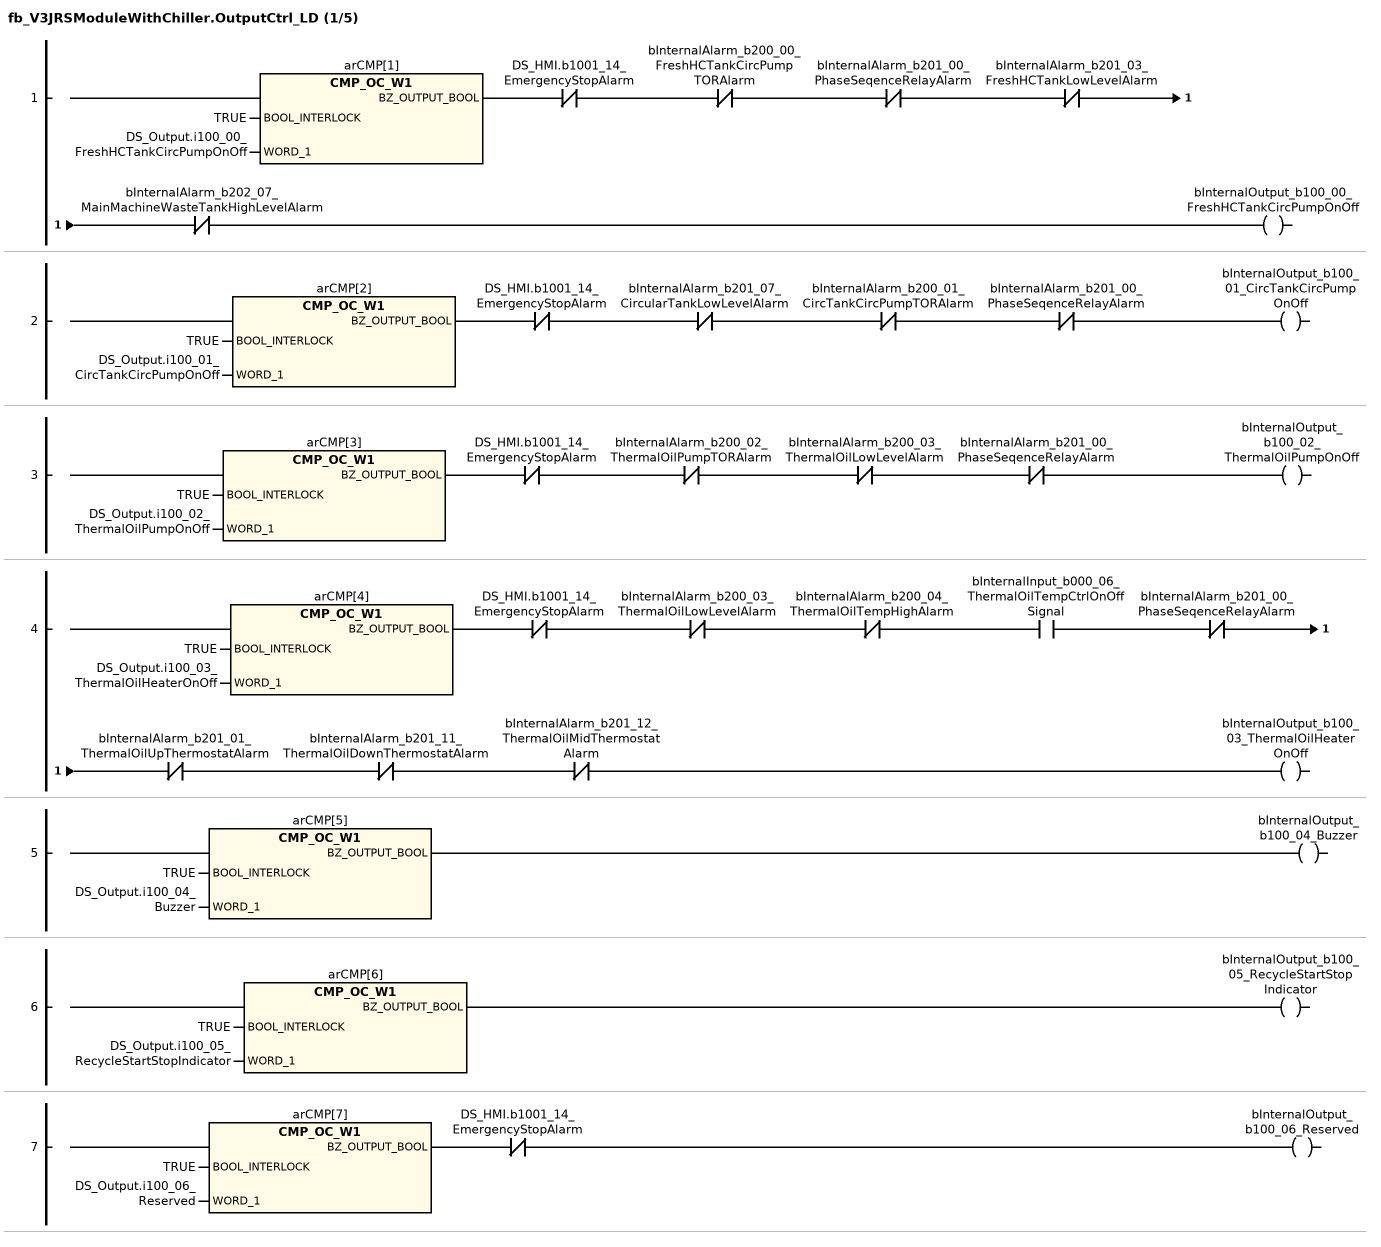
// NETWORK 1
arCMP[1](BOOL_INTERLOCK := TRUE, WORD_1 := DS_Output.i100_00_FreshHCTankCircPumpOnOff); // CMP_OC_W1
bInternalOutput_b100_00_FreshHCTankCircPumpOnOff := arCMP[1].BZ_OUTPUT_BOOL AND NOT DS_HMI.b1001_14_EmergencyStopAlarm AND NOT bInternalAlarm_b200_00_FreshHCTankCircPumpTORAlarm AND NOT bInternalAlarm_b201_00_PhaseSeqenceRelayAlarm AND NOT bInternalAlarm_b201_03_FreshHCTankLowLevelAlarm AND NOT bInternalAlarm_b202_07_MainMachineWasteTankHighLevelAlarm;

// NETWORK 2
arCMP[2](BOOL_INTERLOCK := TRUE, WORD_1 := DS_Output.i100_01_CircTankCircPumpOnOff); // CMP_OC_W1
bInternalOutput_b100_01_CircTankCircPumpOnOff := arCMP[2].BZ_OUTPUT_BOOL AND NOT DS_HMI.b1001_14_EmergencyStopAlarm AND NOT bInternalAlarm_b201_07_CircularTankLowLevelAlarm AND NOT bInternalAlarm_b200_01_CircTankCircPumpTORAlarm AND NOT bInternalAlarm_b201_00_PhaseSeqenceRelayAlarm;

// NETWORK 3
arCMP[3](BOOL_INTERLOCK := TRUE, WORD_1 := DS_Output.i100_02_ThermalOilPumpOnOff); // CMP_OC_W1
bInternalOutput_b100_02_ThermalOilPumpOnOff := arCMP[3].BZ_OUTPUT_BOOL AND NOT DS_HMI.b1001_14_EmergencyStopAlarm AND NOT bInternalAlarm_b200_02_ThermalOilPumpTORAlarm AND NOT bInternalAlarm_b200_03_ThermalOilLowLevelAlarm AND NOT bInternalAlarm_b201_00_PhaseSeqenceRelayAlarm;

// NETWORK 4
arCMP[4](BOOL_INTERLOCK := TRUE, WORD_1 := DS_Output.i100_03_ThermalOilHeaterOnOff); // CMP_OC_W1
bInternalOutput_b100_03_ThermalOilHeaterOnOff := arCMP[4].BZ_OUTPUT_BOOL AND NOT DS_HMI.b1001_14_EmergencyStopAlarm AND NOT bInternalAlarm_b200_03_ThermalOilLowLevelAlarm AND NOT bInternalAlarm_b200_04_ThermalOilTempHighAlarm AND bInternalInput_b000_06_ThermalOilTempCtrlOnOffSignal AND NOT bInternalAlarm_b201_00_PhaseSeqenceRelayAlarm AND NOT bInternalAlarm_b201_01_ThermalOilUpThermostatAlarm AND NOT bInternalAlarm_b201_11_ThermalOilDownThermostatAlarm AND NOT bInternalAlarm_b201_12_ThermalOilMidThermostatAlarm;

// NETWORK 5
arCMP[5](BOOL_INTERLOCK := TRUE, WORD_1 := DS_Output.i100_04_Buzzer); // CMP_OC_W1
bInternalOutput_b100_04_Buzzer := arCMP[5].BZ_OUTPUT_BOOL;

// NETWORK 6
arCMP[6](BOOL_INTERLOCK := TRUE, WORD_1 := DS_Output.i100_05_RecycleStartStopIndicator); // CMP_OC_W1
bInternalOutput_b100_05_RecycleStartStopIndicator := arCMP[6].BZ_OUTPUT_BOOL;

// NETWORK 7
arCMP[7](BOOL_INTERLOCK := TRUE, WORD_1 := DS_Output.i100_06_Reserved); // CMP_OC_W1
bInternalOutput_b100_06_Reserved := arCMP[7].BZ_OUTPUT_BOOL AND NOT DS_HMI.b1001_14_EmergencyStopAlarm;

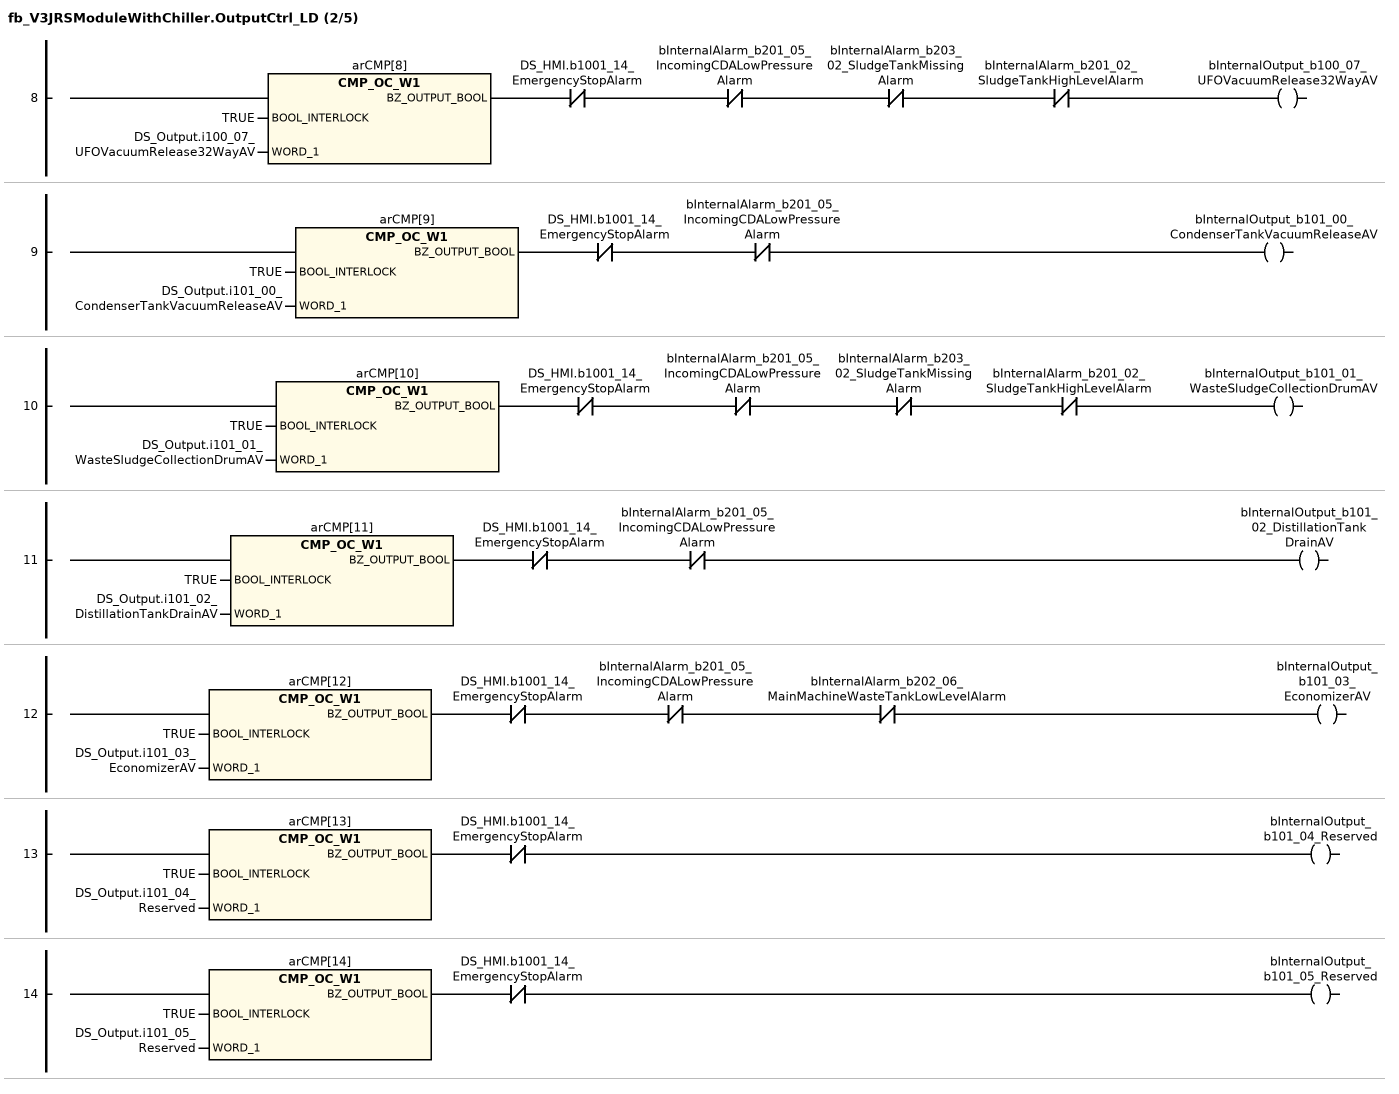
// NETWORK 8
arCMP[8](BOOL_INTERLOCK := TRUE, WORD_1 := DS_Output.i100_07_UFOVacuumRelease32WayAV); // CMP_OC_W1
bInternalOutput_b100_07_UFOVacuumRelease32WayAV := arCMP[8].BZ_OUTPUT_BOOL AND NOT DS_HMI.b1001_14_EmergencyStopAlarm AND NOT bInternalAlarm_b201_05_IncomingCDALowPressureAlarm AND NOT bInternalAlarm_b203_02_SludgeTankMissingAlarm AND NOT bInternalAlarm_b201_02_SludgeTankHighLevelAlarm;

// NETWORK 9
arCMP[9](BOOL_INTERLOCK := TRUE, WORD_1 := DS_Output.i101_00_CondenserTankVacuumReleaseAV); // CMP_OC_W1
bInternalOutput_b101_00_CondenserTankVacuumReleaseAV := arCMP[9].BZ_OUTPUT_BOOL AND NOT DS_HMI.b1001_14_EmergencyStopAlarm AND NOT bInternalAlarm_b201_05_IncomingCDALowPressureAlarm;

// NETWORK 10
arCMP[10](BOOL_INTERLOCK := TRUE, WORD_1 := DS_Output.i101_01_WasteSludgeCollectionDrumAV); // CMP_OC_W1
bInternalOutput_b101_01_WasteSludgeCollectionDrumAV := arCMP[10].BZ_OUTPUT_BOOL AND NOT DS_HMI.b1001_14_EmergencyStopAlarm AND NOT bInternalAlarm_b201_05_IncomingCDALowPressureAlarm AND NOT bInternalAlarm_b203_02_SludgeTankMissingAlarm AND NOT bInternalAlarm_b201_02_SludgeTankHighLevelAlarm;

// NETWORK 11
arCMP[11](BOOL_INTERLOCK := TRUE, WORD_1 := DS_Output.i101_02_DistillationTankDrainAV); // CMP_OC_W1
bInternalOutput_b101_02_DistillationTankDrainAV := arCMP[11].BZ_OUTPUT_BOOL AND NOT DS_HMI.b1001_14_EmergencyStopAlarm AND NOT bInternalAlarm_b201_05_IncomingCDALowPressureAlarm;

// NETWORK 12
arCMP[12](BOOL_INTERLOCK := TRUE, WORD_1 := DS_Output.i101_03_EconomizerAV); // CMP_OC_W1
bInternalOutput_b101_03_EconomizerAV := arCMP[12].BZ_OUTPUT_BOOL AND NOT DS_HMI.b1001_14_EmergencyStopAlarm AND NOT bInternalAlarm_b201_05_IncomingCDALowPressureAlarm AND NOT bInternalAlarm_b202_06_MainMachineWasteTankLowLevelAlarm;

// NETWORK 13
arCMP[13](BOOL_INTERLOCK := TRUE, WORD_1 := DS_Output.i101_04_Reserved); // CMP_OC_W1
bInternalOutput_b101_04_Reserved := arCMP[13].BZ_OUTPUT_BOOL AND NOT DS_HMI.b1001_14_EmergencyStopAlarm;

// NETWORK 14
arCMP[14](BOOL_INTERLOCK := TRUE, WORD_1 := DS_Output.i101_05_Reserved); // CMP_OC_W1
bInternalOutput_b101_05_Reserved := arCMP[14].BZ_OUTPUT_BOOL AND NOT DS_HMI.b1001_14_EmergencyStopAlarm;

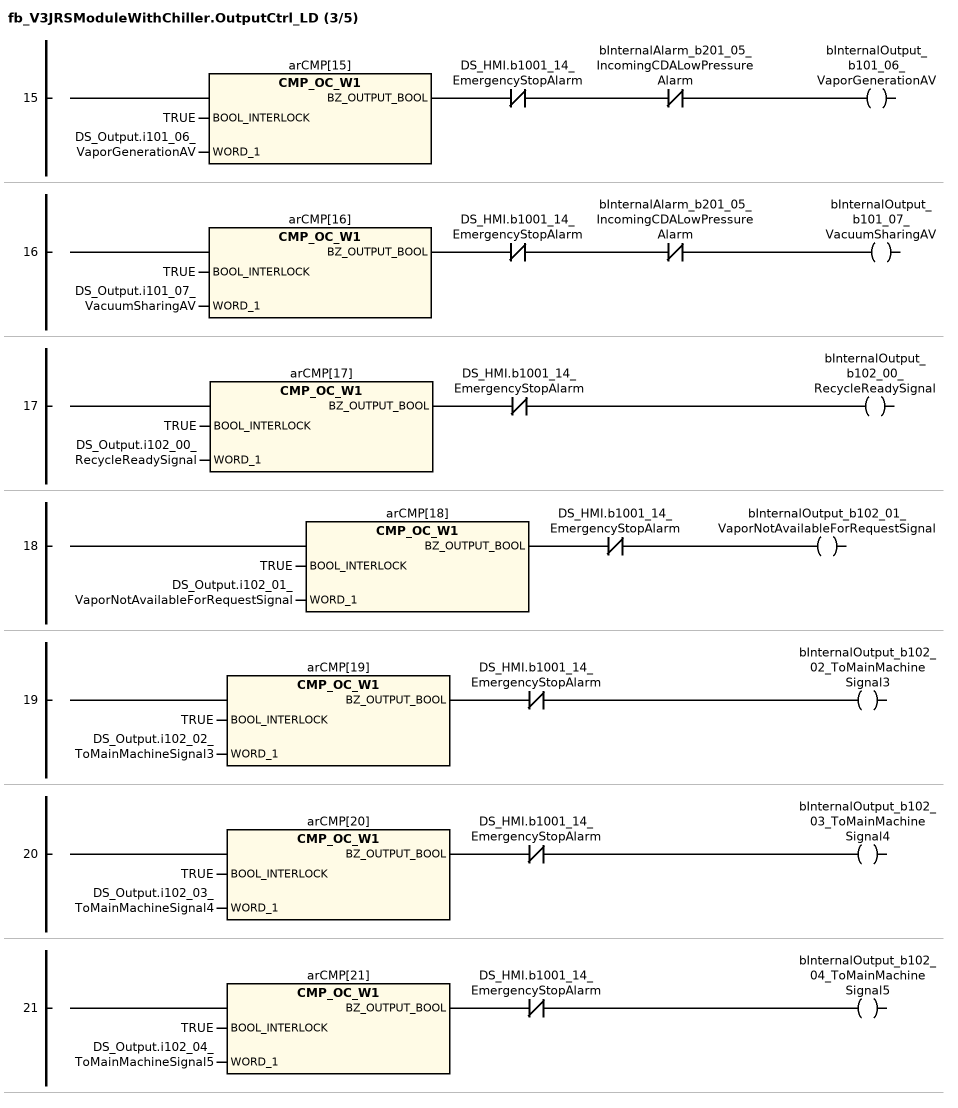
// NETWORK 15
arCMP[15](BOOL_INTERLOCK := TRUE, WORD_1 := DS_Output.i101_06_VaporGenerationAV); // CMP_OC_W1
bInternalOutput_b101_06_VaporGenerationAV := arCMP[15].BZ_OUTPUT_BOOL AND NOT DS_HMI.b1001_14_EmergencyStopAlarm AND NOT bInternalAlarm_b201_05_IncomingCDALowPressureAlarm;

// NETWORK 16
arCMP[16](BOOL_INTERLOCK := TRUE, WORD_1 := DS_Output.i101_07_VacuumSharingAV); // CMP_OC_W1
bInternalOutput_b101_07_VacuumSharingAV := arCMP[16].BZ_OUTPUT_BOOL AND NOT DS_HMI.b1001_14_EmergencyStopAlarm AND NOT bInternalAlarm_b201_05_IncomingCDALowPressureAlarm;

// NETWORK 17
arCMP[17](BOOL_INTERLOCK := TRUE, WORD_1 := DS_Output.i102_00_RecycleReadySignal); // CMP_OC_W1
bInternalOutput_b102_00_RecycleReadySignal := arCMP[17].BZ_OUTPUT_BOOL AND NOT DS_HMI.b1001_14_EmergencyStopAlarm;

// NETWORK 18
arCMP[18](BOOL_INTERLOCK := TRUE, WORD_1 := DS_Output.i102_01_VaporNotAvailableForRequestSignal); // CMP_OC_W1
bInternalOutput_b102_01_VaporNotAvailableForRequestSignal := arCMP[18].BZ_OUTPUT_BOOL AND NOT DS_HMI.b1001_14_EmergencyStopAlarm;

// NETWORK 19
arCMP[19](BOOL_INTERLOCK := TRUE, WORD_1 := DS_Output.i102_02_ToMainMachineSignal3); // CMP_OC_W1
bInternalOutput_b102_02_ToMainMachineSignal3 := arCMP[19].BZ_OUTPUT_BOOL AND NOT DS_HMI.b1001_14_EmergencyStopAlarm;

// NETWORK 20
arCMP[20](BOOL_INTERLOCK := TRUE, WORD_1 := DS_Output.i102_03_ToMainMachineSignal4); // CMP_OC_W1
bInternalOutput_b102_03_ToMainMachineSignal4 := arCMP[20].BZ_OUTPUT_BOOL AND NOT DS_HMI.b1001_14_EmergencyStopAlarm;

// NETWORK 21
arCMP[21](BOOL_INTERLOCK := TRUE, WORD_1 := DS_Output.i102_04_ToMainMachineSignal5); // CMP_OC_W1
bInternalOutput_b102_04_ToMainMachineSignal5 := arCMP[21].BZ_OUTPUT_BOOL AND NOT DS_HMI.b1001_14_EmergencyStopAlarm;

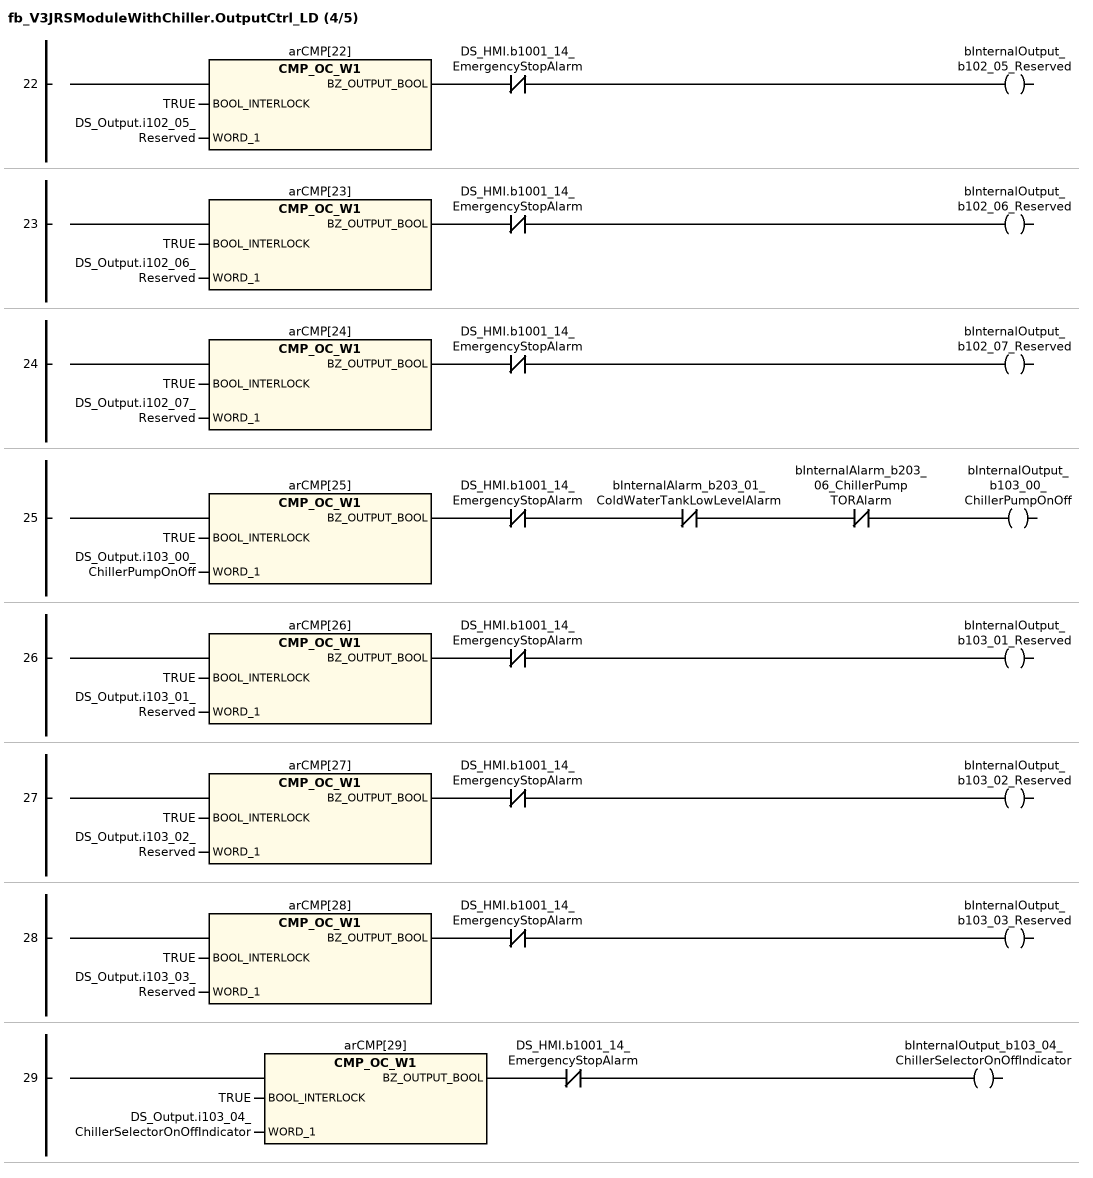
// NETWORK 22
arCMP[22](BOOL_INTERLOCK := TRUE, WORD_1 := DS_Output.i102_05_Reserved); // CMP_OC_W1
bInternalOutput_b102_05_Reserved := arCMP[22].BZ_OUTPUT_BOOL AND NOT DS_HMI.b1001_14_EmergencyStopAlarm;

// NETWORK 23
arCMP[23](BOOL_INTERLOCK := TRUE, WORD_1 := DS_Output.i102_06_Reserved); // CMP_OC_W1
bInternalOutput_b102_06_Reserved := arCMP[23].BZ_OUTPUT_BOOL AND NOT DS_HMI.b1001_14_EmergencyStopAlarm;

// NETWORK 24
arCMP[24](BOOL_INTERLOCK := TRUE, WORD_1 := DS_Output.i102_07_Reserved); // CMP_OC_W1
bInternalOutput_b102_07_Reserved := arCMP[24].BZ_OUTPUT_BOOL AND NOT DS_HMI.b1001_14_EmergencyStopAlarm;

// NETWORK 25
arCMP[25](BOOL_INTERLOCK := TRUE, WORD_1 := DS_Output.i103_00_ChillerPumpOnOff); // CMP_OC_W1
bInternalOutput_b103_00_ChillerPumpOnOff := arCMP[25].BZ_OUTPUT_BOOL AND NOT DS_HMI.b1001_14_EmergencyStopAlarm AND NOT bInternalAlarm_b203_01_ColdWaterTankLowLevelAlarm AND NOT bInternalAlarm_b203_06_ChillerPumpTORAlarm;

// NETWORK 26
arCMP[26](BOOL_INTERLOCK := TRUE, WORD_1 := DS_Output.i103_01_Reserved); // CMP_OC_W1
bInternalOutput_b103_01_Reserved := arCMP[26].BZ_OUTPUT_BOOL AND NOT DS_HMI.b1001_14_EmergencyStopAlarm;

// NETWORK 27
arCMP[27](BOOL_INTERLOCK := TRUE, WORD_1 := DS_Output.i103_02_Reserved); // CMP_OC_W1
bInternalOutput_b103_02_Reserved := arCMP[27].BZ_OUTPUT_BOOL AND NOT DS_HMI.b1001_14_EmergencyStopAlarm;

// NETWORK 28
arCMP[28](BOOL_INTERLOCK := TRUE, WORD_1 := DS_Output.i103_03_Reserved); // CMP_OC_W1
bInternalOutput_b103_03_Reserved := arCMP[28].BZ_OUTPUT_BOOL AND NOT DS_HMI.b1001_14_EmergencyStopAlarm;

// NETWORK 29
arCMP[29](BOOL_INTERLOCK := TRUE, WORD_1 := DS_Output.i103_04_ChillerSelectorOnOffIndicator); // CMP_OC_W1
bInternalOutput_b103_04_ChillerSelectorOnOffIndicator := arCMP[29].BZ_OUTPUT_BOOL AND NOT DS_HMI.b1001_14_EmergencyStopAlarm;

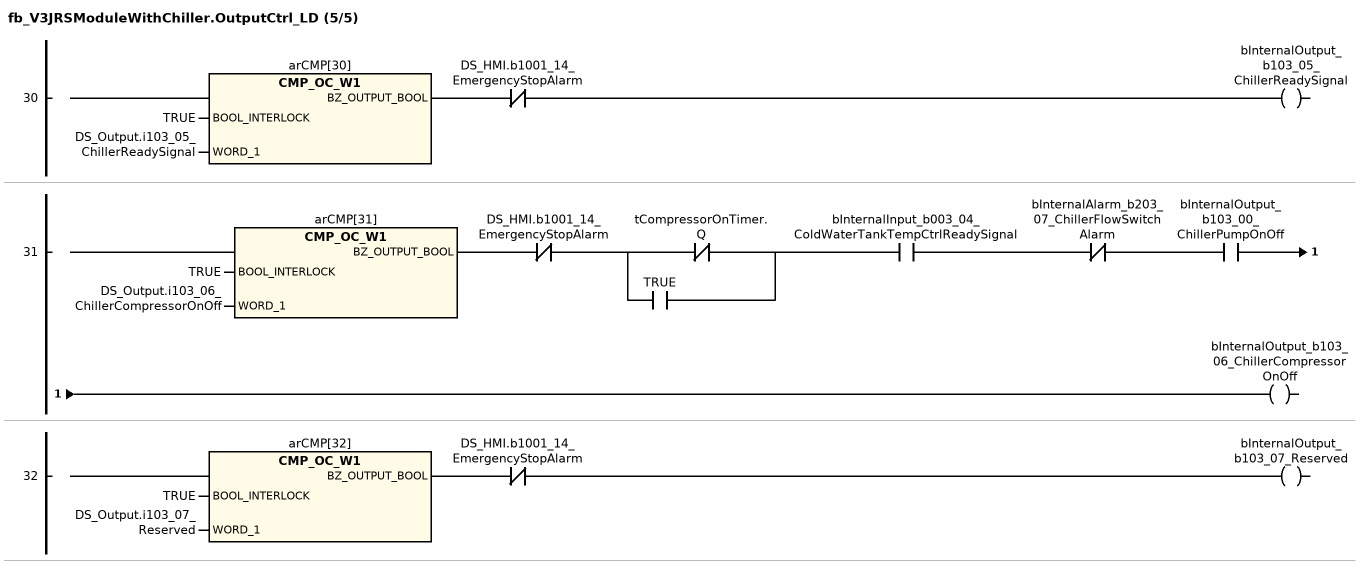
// NETWORK 30
arCMP[30](BOOL_INTERLOCK := TRUE, WORD_1 := DS_Output.i103_05_ChillerReadySignal); // CMP_OC_W1
bInternalOutput_b103_05_ChillerReadySignal := arCMP[30].BZ_OUTPUT_BOOL AND NOT DS_HMI.b1001_14_EmergencyStopAlarm;

// NETWORK 31
arCMP[31](BOOL_INTERLOCK := TRUE, WORD_1 := DS_Output.i103_06_ChillerCompressorOnOff); // CMP_OC_W1
bInternalOutput_b103_06_ChillerCompressorOnOff := (arCMP[31].BZ_OUTPUT_BOOL AND NOT DS_HMI.b1001_14_EmergencyStopAlarm AND (NOT tCompressorOnTimer.Q OR TRUE)) AND bInternalInput_b003_04_ColdWaterTankTempCtrlReadySignal AND NOT bInternalAlarm_b203_07_ChillerFlowSwitchAlarm AND bInternalOutput_b103_00_ChillerPumpOnOff;

// NETWORK 32
arCMP[32](BOOL_INTERLOCK := TRUE, WORD_1 := DS_Output.i103_07_Reserved); // CMP_OC_W1
bInternalOutput_b103_07_Reserved := arCMP[32].BZ_OUTPUT_BOOL AND NOT DS_HMI.b1001_14_EmergencyStopAlarm;
END_ACTION

ACTION SystemRestore_LD:
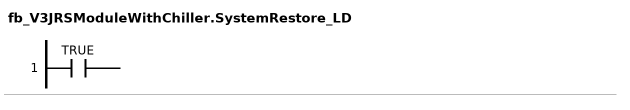
// NETWORK 1
END_ACTION

ACTION ThermalOilChangeHRMeter_ST:
	(*ThermalOilChange Hour Meter Counting*)
	IF bInternalOutput_b100_02_ThermalOilPumpOnOff AND t1SecCPRE.Q THEN

		DS_HMI.iD242_ThermalOilChangeHMeterPV_Sec := DS_HMI.iD242_ThermalOilChangeHMeterPV_Sec +1;
	
		IF DS_HMI.iD242_ThermalOilChangeHMeterPV_Sec > 59 THEN
			DS_HMI.iD241_ThermalOilChangeHMeterPV_Min := DS_HMI.iD241_ThermalOilChangeHMeterPV_Min +1;
			DS_HMI.iD242_ThermalOilChangeHMeterPV_Sec := 0;
		END_IF
	
		IF DS_HMI.iD241_ThermalOilChangeHMeterPV_Min > 59 THEN
			DS_HMI.iD240_ThermalOilChangeHMeterPV_Hour := DS_HMI.iD240_ThermalOilChangeHMeterPV_Hour +1;
			DS_HMI.iD241_ThermalOilChangeHMeterPV_Min := 0;
		END_IF

	END_IF
	

	(*ThermalOilChange Hour Meter Warning and Alarm*)
	IF DS_HMI.iD240_ThermalOilChangeHMeterPV_Hour >= DS_HMI.iD251_ThermalOilChangeAlarmSV_Hour THEN
	DS_HMI.b1040_00_ThermalOilChangeHMeterAlarm := TRUE;
	ELSE
	DS_HMI.b1040_00_ThermalOilChangeHMeterAlarm := FALSE;
	END_IF

	IF DS_HMI.iD240_ThermalOilChangeHMeterPV_Hour >= DS_HMI.iD250_ThermalOilChangeWarningSV_Hour THEN
	DS_HMI.b1040_02_ThermalOiChangeWarning := TRUE;
	ELSE
	DS_HMI.b1040_02_ThermalOiChangeWarning := FALSE;
	END_IF

	(*ThermalOilChange Hour Meter Reset*)
	tThermalOilChangeResetPBTimer(IN:=DS_HMI.b1040_01_ThermalOilChangeHMeterResetPB , PT:=t#3s , Q=> , ET=> );
	IF tThermalOilChangeResetPBTimer.Q THEN

		DS_HMI.iD242_ThermalOilChangeHMeterPV_Sec	:= 0;
		DS_HMI.iD241_ThermalOilChangeHMeterPV_Min	:= 0;
		DS_HMI.iD240_ThermalOilChangeHMeterPV_Hour	:= 0;
	END_IF
END_ACTION

ACTION Z_BuiltInTempCtrl_LD:
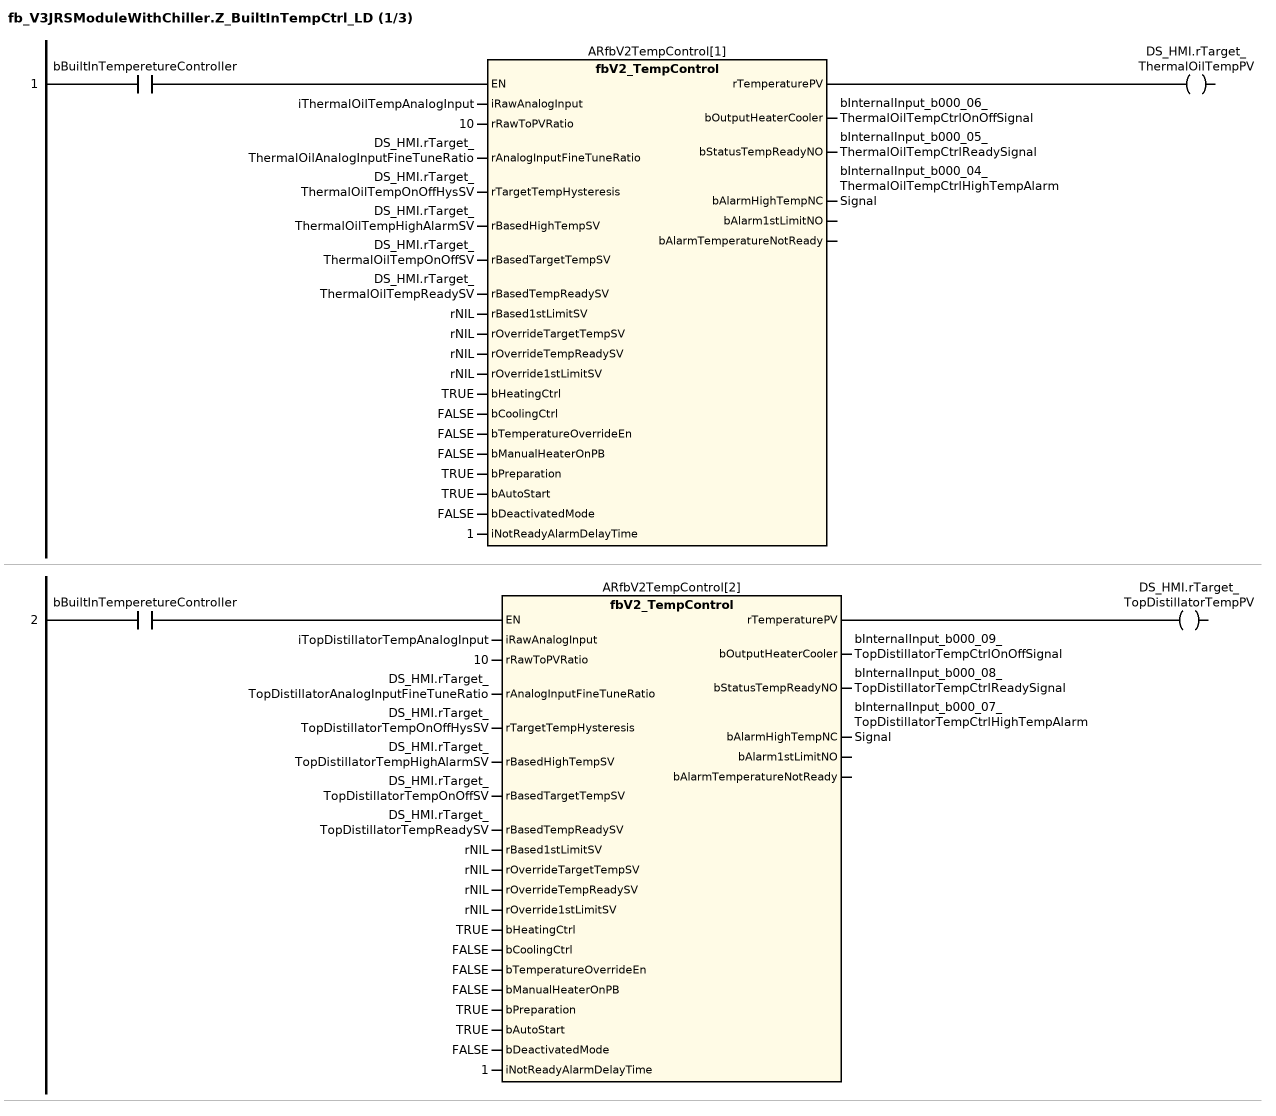
// NETWORK 1
IF bBuiltInTemperetureController THEN
    ARfbV2TempControl[1](
        iRawAnalogInput := iThermalOilTempAnalogInput,
        rRawToPVRatio := 10,
        rAnalogInputFineTuneRatio := DS_HMI.rTarget_ThermalOilAnalogInputFineTuneRatio,
        rTargetTempHysteresis := DS_HMI.rTarget_ThermalOilTempOnOffHysSV,
        rBasedHighTempSV := DS_HMI.rTarget_ThermalOilTempHighAlarmSV,
        rBasedTargetTempSV := DS_HMI.rTarget_ThermalOilTempOnOffSV,
        rBasedTempReadySV := DS_HMI.rTarget_ThermalOilTempReadySV,
        rBased1stLimitSV := rNIL,
        rOverrideTargetTempSV := rNIL,
        rOverrideTempReadySV := rNIL,
        rOverride1stLimitSV := rNIL,
        bHeatingCtrl := TRUE,
        bCoolingCtrl := FALSE,
        bTemperatureOverrideEn := FALSE,
        bManualHeaterOnPB := FALSE,
        bPreparation := TRUE,
        bAutoStart := TRUE,
        bDeactivatedMode := FALSE,
        iNotReadyAlarmDelayTime := 1,
        bOutputHeaterCooler => bInternalInput_b000_06_ThermalOilTempCtrlOnOffSignal,
        bStatusTempReadyNO => bInternalInput_b000_05_ThermalOilTempCtrlReadySignal,
        bAlarmHighTempNC => bInternalInput_b000_04_ThermalOilTempCtrlHighTempAlarmSignal); // fbV2_TempControl
END_IF
DS_HMI.rTarget_ThermalOilTempPV := ARfbV2TempControl[1].rTemperaturePV;

// NETWORK 2
IF bBuiltInTemperetureController THEN
    ARfbV2TempControl[2](
        iRawAnalogInput := iTopDistillatorTempAnalogInput,
        rRawToPVRatio := 10,
        rAnalogInputFineTuneRatio := DS_HMI.rTarget_TopDistillatorAnalogInputFineTuneRatio,
        rTargetTempHysteresis := DS_HMI.rTarget_TopDistillatorTempOnOffHysSV,
        rBasedHighTempSV := DS_HMI.rTarget_TopDistillatorTempHighAlarmSV,
        rBasedTargetTempSV := DS_HMI.rTarget_TopDistillatorTempOnOffSV,
        rBasedTempReadySV := DS_HMI.rTarget_TopDistillatorTempReadySV,
        rBased1stLimitSV := rNIL,
        rOverrideTargetTempSV := rNIL,
        rOverrideTempReadySV := rNIL,
        rOverride1stLimitSV := rNIL,
        bHeatingCtrl := TRUE,
        bCoolingCtrl := FALSE,
        bTemperatureOverrideEn := FALSE,
        bManualHeaterOnPB := FALSE,
        bPreparation := TRUE,
        bAutoStart := TRUE,
        bDeactivatedMode := FALSE,
        iNotReadyAlarmDelayTime := 1,
        bOutputHeaterCooler => bInternalInput_b000_09_TopDistillatorTempCtrlOnOffSignal,
        bStatusTempReadyNO => bInternalInput_b000_08_TopDistillatorTempCtrlReadySignal,
        bAlarmHighTempNC => bInternalInput_b000_07_TopDistillatorTempCtrlHighTempAlarmSignal); // fbV2_TempControl
END_IF
DS_HMI.rTarget_TopDistillatorTempPV := ARfbV2TempControl[2].rTemperaturePV;

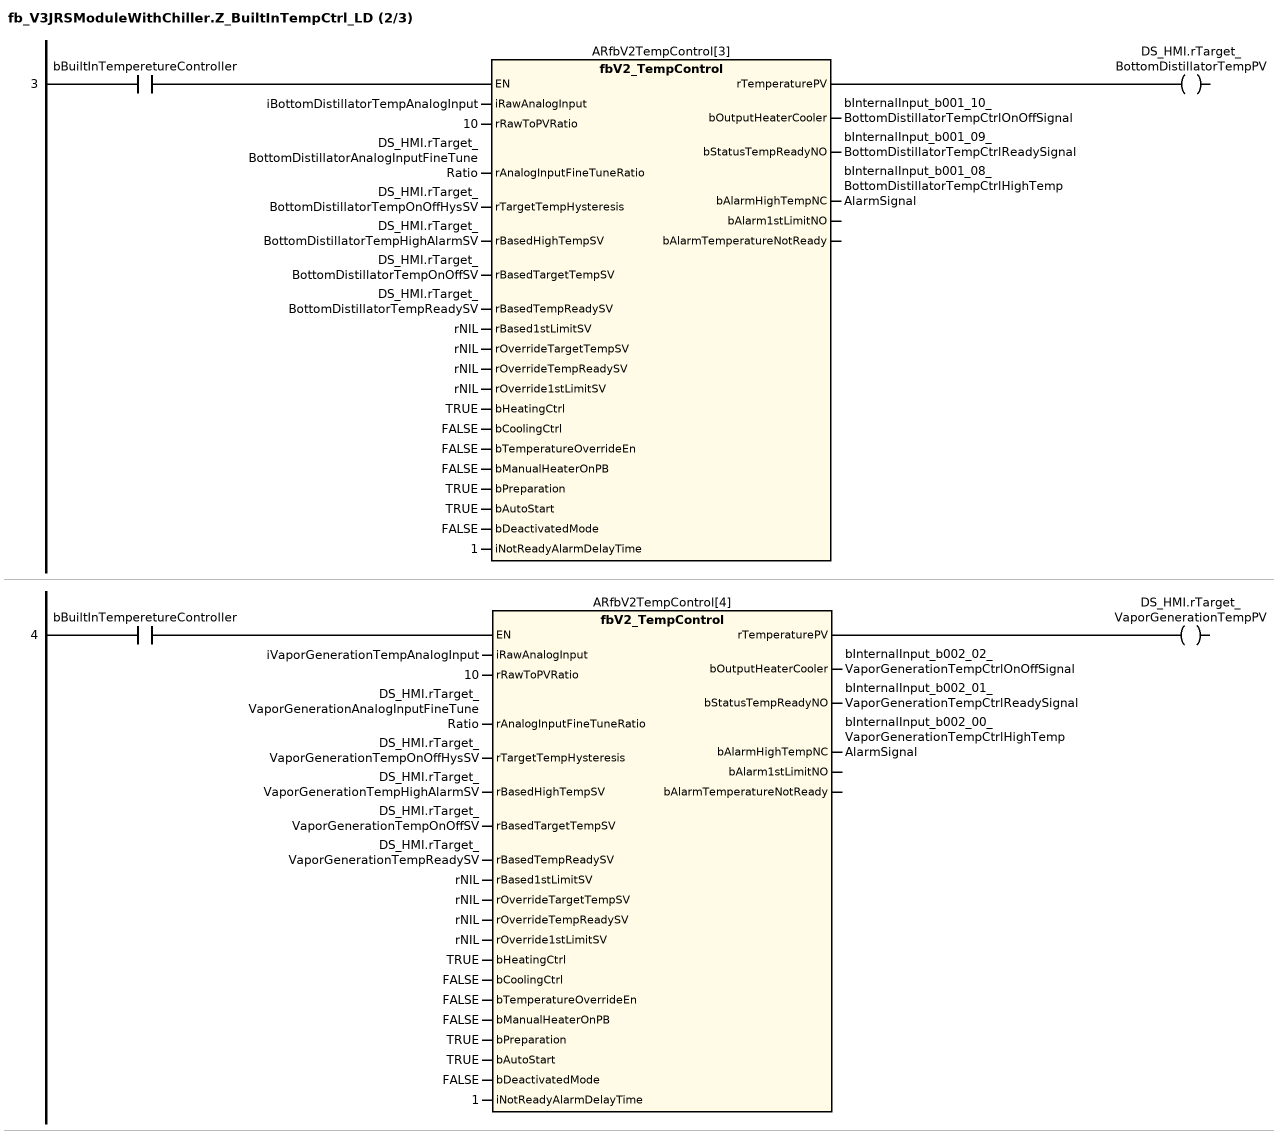
// NETWORK 3
IF bBuiltInTemperetureController THEN
    ARfbV2TempControl[3](
        iRawAnalogInput := iBottomDistillatorTempAnalogInput,
        rRawToPVRatio := 10,
        rAnalogInputFineTuneRatio := DS_HMI.rTarget_BottomDistillatorAnalogInputFineTuneRatio,
        rTargetTempHysteresis := DS_HMI.rTarget_BottomDistillatorTempOnOffHysSV,
        rBasedHighTempSV := DS_HMI.rTarget_BottomDistillatorTempHighAlarmSV,
        rBasedTargetTempSV := DS_HMI.rTarget_BottomDistillatorTempOnOffSV,
        rBasedTempReadySV := DS_HMI.rTarget_BottomDistillatorTempReadySV,
        rBased1stLimitSV := rNIL,
        rOverrideTargetTempSV := rNIL,
        rOverrideTempReadySV := rNIL,
        rOverride1stLimitSV := rNIL,
        bHeatingCtrl := TRUE,
        bCoolingCtrl := FALSE,
        bTemperatureOverrideEn := FALSE,
        bManualHeaterOnPB := FALSE,
        bPreparation := TRUE,
        bAutoStart := TRUE,
        bDeactivatedMode := FALSE,
        iNotReadyAlarmDelayTime := 1,
        bOutputHeaterCooler => bInternalInput_b001_10_BottomDistillatorTempCtrlOnOffSignal,
        bStatusTempReadyNO => bInternalInput_b001_09_BottomDistillatorTempCtrlReadySignal,
        bAlarmHighTempNC => bInternalInput_b001_08_BottomDistillatorTempCtrlHighTempAlarmSignal); // fbV2_TempControl
END_IF
DS_HMI.rTarget_BottomDistillatorTempPV := ARfbV2TempControl[3].rTemperaturePV;

// NETWORK 4
IF bBuiltInTemperetureController THEN
    ARfbV2TempControl[4](
        iRawAnalogInput := iVaporGenerationTempAnalogInput,
        rRawToPVRatio := 10,
        rAnalogInputFineTuneRatio := DS_HMI.rTarget_VaporGenerationAnalogInputFineTuneRatio,
        rTargetTempHysteresis := DS_HMI.rTarget_VaporGenerationTempOnOffHysSV,
        rBasedHighTempSV := DS_HMI.rTarget_VaporGenerationTempHighAlarmSV,
        rBasedTargetTempSV := DS_HMI.rTarget_VaporGenerationTempOnOffSV,
        rBasedTempReadySV := DS_HMI.rTarget_VaporGenerationTempReadySV,
        rBased1stLimitSV := rNIL,
        rOverrideTargetTempSV := rNIL,
        rOverrideTempReadySV := rNIL,
        rOverride1stLimitSV := rNIL,
        bHeatingCtrl := TRUE,
        bCoolingCtrl := FALSE,
        bTemperatureOverrideEn := FALSE,
        bManualHeaterOnPB := FALSE,
        bPreparation := TRUE,
        bAutoStart := TRUE,
        bDeactivatedMode := FALSE,
        iNotReadyAlarmDelayTime := 1,
        bOutputHeaterCooler => bInternalInput_b002_02_VaporGenerationTempCtrlOnOffSignal,
        bStatusTempReadyNO => bInternalInput_b002_01_VaporGenerationTempCtrlReadySignal,
        bAlarmHighTempNC => bInternalInput_b002_00_VaporGenerationTempCtrlHighTempAlarmSignal); // fbV2_TempControl
END_IF
DS_HMI.rTarget_VaporGenerationTempPV := ARfbV2TempControl[4].rTemperaturePV;

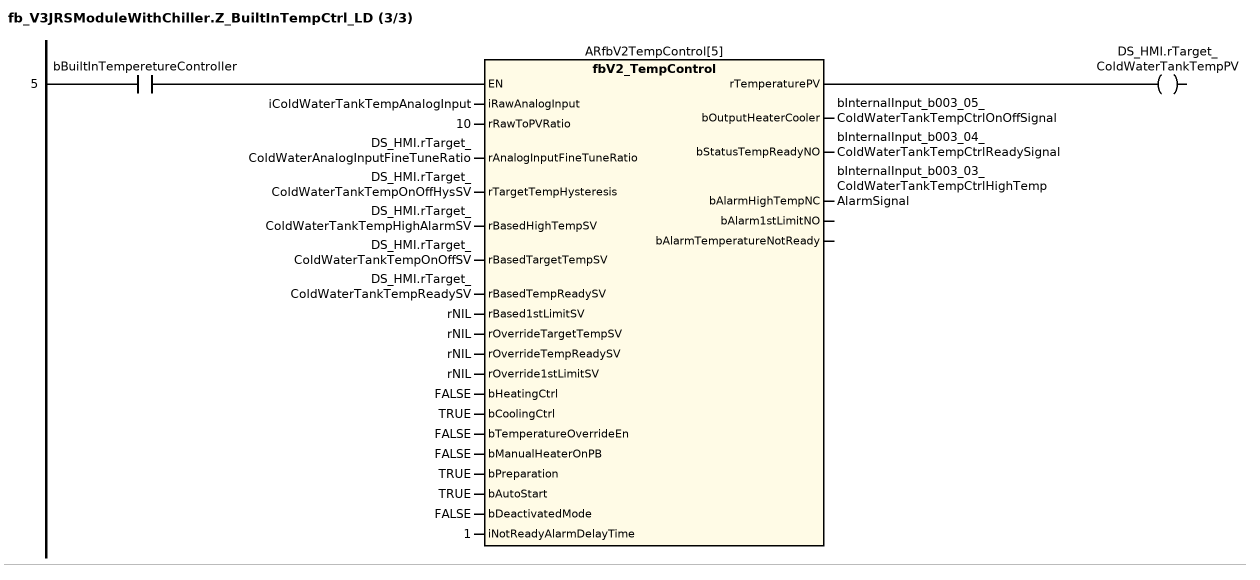
// NETWORK 5
IF bBuiltInTemperetureController THEN
    ARfbV2TempControl[5](
        iRawAnalogInput := iColdWaterTankTempAnalogInput,
        rRawToPVRatio := 10,
        rAnalogInputFineTuneRatio := DS_HMI.rTarget_ColdWaterAnalogInputFineTuneRatio,
        rTargetTempHysteresis := DS_HMI.rTarget_ColdWaterTankTempOnOffHysSV,
        rBasedHighTempSV := DS_HMI.rTarget_ColdWaterTankTempHighAlarmSV,
        rBasedTargetTempSV := DS_HMI.rTarget_ColdWaterTankTempOnOffSV,
        rBasedTempReadySV := DS_HMI.rTarget_ColdWaterTankTempReadySV,
        rBased1stLimitSV := rNIL,
        rOverrideTargetTempSV := rNIL,
        rOverrideTempReadySV := rNIL,
        rOverride1stLimitSV := rNIL,
        bHeatingCtrl := FALSE,
        bCoolingCtrl := TRUE,
        bTemperatureOverrideEn := FALSE,
        bManualHeaterOnPB := FALSE,
        bPreparation := TRUE,
        bAutoStart := TRUE,
        bDeactivatedMode := FALSE,
        iNotReadyAlarmDelayTime := 1,
        bOutputHeaterCooler => bInternalInput_b003_05_ColdWaterTankTempCtrlOnOffSignal,
        bStatusTempReadyNO => bInternalInput_b003_04_ColdWaterTankTempCtrlReadySignal,
        bAlarmHighTempNC => bInternalInput_b003_03_ColdWaterTankTempCtrlHighTempAlarmSignal); // fbV2_TempControl
END_IF
DS_HMI.rTarget_ColdWaterTankTempPV := ARfbV2TempControl[5].rTemperaturePV;
END_ACTION

ACTION Z_BuiltInTempCtrl_ST:
	IF NOT bBuiltInTemperetureController THEN
	bInternalInput_b000_04_ThermalOilTempCtrlHighTempAlarmSignal 		:= 	DS_Input.b000_04_ThermalOilTempCtrlHighTempAlarmSignal;
	bInternalInput_b000_05_ThermalOilTempCtrlReadySignal			 	:= 	DS_Input.b000_05_ThermalOilTempCtrlReadySignal;
	bInternalInput_b000_06_ThermalOilTempCtrlOnOffSignal  				:= 	DS_Input.b000_06_ThermalOilTempCtrlOnOffSignal ;
	bInternalInput_b000_07_TopDistillatorTempCtrlHighTempAlarmSignal 		:= 	DS_Input.b000_07_TopDistillatorTempCtrlHighTempAlarmSignal;
	bInternalInput_b000_08_TopDistillatorTempCtrlReadySignal 				:= 	DS_Input.b000_08_TopDistillatorTempCtrlReadySignal;
	bInternalInput_b000_09_TopDistillatorTempCtrlOnOffSignal  				:= 	DS_Input.b000_09_TopDistillatorTempCtrlOnOffSignal ;
	bInternalInput_b001_08_BottomDistillatorTempCtrlHighTempAlarmSignal 	:= 	DS_Input.b001_08_BottomDistillatorTempCtrlHighTempAlarmSignal;
	bInternalInput_b001_09_BottomDistillatorTempCtrlReadySignal 			:= 	DS_Input.b001_09_BottomDistillatorTempCtrlReadySignal;
	bInternalInput_b001_10_BottomDistillatorTempCtrlOnOffSignal  			:= 	DS_Input.b001_10_BottomDistillatorTempCtrlOnOffSignal ;
	bInternalInput_b002_00_VaporGenerationTempCtrlHighTempAlarmSignal 	:= 	DS_Input.b002_00_VaporGenerationTempCtrlHighTempAlarmSignal;
	bInternalInput_b002_01_VaporGenerationTempCtrlReadySignal 			:= 	DS_Input.b002_01_VaporGenerationTempCtrlReadySignal;
	bInternalInput_b002_02_VaporGenerationTempCtrlOnOffSignal 			:= 	DS_Input.b002_02_VaporGenerationTempCtrlOnOffSignal;
	bInternalInput_b003_03_ColdWaterTankTempCtrlHighTempAlarmSignal 	:= 	DS_Input.b003_03_ColdWaterTankTempCtrlHighTempAlarmSignal;
	bInternalInput_b003_04_ColdWaterTankTempCtrlReadySignal 			:= 	DS_Input.b003_04_ColdWaterTankTempCtrlReadySignal;
	bInternalInput_b003_05_ColdWaterTankTempCtrlOnOffSignal 			:= 	DS_Input.b003_05_ColdWaterTankTempCtrlOnOffSignal;

	ELSE

	Z_BuiltInTempCtrl_LD();
	END_IF

(*
	iThermalOilTempAnalogInput;			AT %I* : INT;
	iTopDistillatorTempAnalogInput;			AT %I* : INT;
	iBottomDistillatorTempAnalogInput;		AT %I* : INT;
	iVaporGenerationTempAnalogInput;		AT %I* : INT;
	iColdWaterTankTempAnalogInput; 		AT %I* : INT;


*)
END_ACTION

ACTION Z_BuiltInVacuumCtrl_LD:
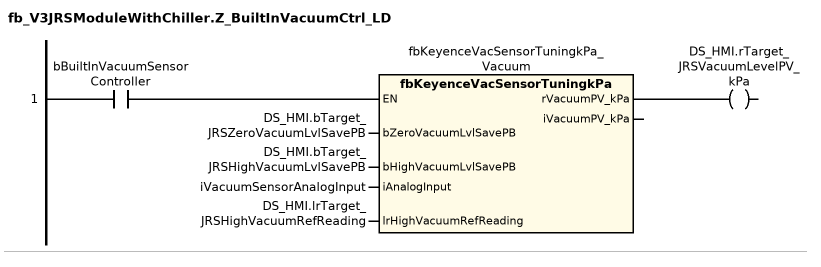
// NETWORK 1
IF bBuiltInVacuumSensorController THEN
    fbKeyenceVacSensorTuningkPa_Vacuum(
        bZeroVacuumLvlSavePB := DS_HMI.bTarget_JRSZeroVacuumLvlSavePB,
        bHighVacuumLvlSavePB := DS_HMI.bTarget_JRSHighVacuumLvlSavePB,
        iAnalogInput := iVacuumSensorAnalogInput,
        lrHighVacuumRefReading := DS_HMI.lrTarget_JRSHighVacuumRefReading); // fbKeyenceVacSensorTuningkPa
END_IF
DS_HMI.rTarget_JRSVacuumLevelPV_kPa := fbKeyenceVacSensorTuningkPa_Vacuum.rVacuumPV_kPa;
END_ACTION

ACTION Z_BuiltInVacuumCtrl_ST:
	IF NOT bBuiltInVacuumSensorController THEN

		bInternalInput_b001_04_VacuumNotAchieveSignal 		:= 	DS_Input.b001_04_VacuumNotAchieveSignal;

	ELSE

		Z_BuiltInVacuumCtrl_LD();

		bVacuumAchieveFlag := FALSE;

		(*Compare and trigger output*)
		IF bBuiltInVacuumNegativeSignal THEN

			IF DS_HMI.rTarget_JRSVacuumLevelPV_kPa <= DS_HMI.rTarget_JRSVacuumLevelSV_kPa THEN
				bVacuumAchieveFlag := TRUE;
			END_IF

		ELSE

			IF DS_HMI.rTarget_JRSVacuumLevelPV_kPa >= DS_HMI.rTarget_JRSVacuumLevelSV_kPa THEN
				bVacuumAchieveFlag := TRUE;
			END_IF

		END_IF

		bInternalInput_b001_04_VacuumNotAchieveSignal := NOT bVacuumAchieveFlag;


	END_IF
END_ACTION

ACTION Z_Mapping:
		(*Mapping - Alarm*)
		DS_Alarm.b200_00_FreshHCTankCircPumpTORAlarm  := bInternalAlarm_b200_00_FreshHCTankCircPumpTORAlarm ;
		DS_Alarm.b200_01_CircTankCircPumpTORAlarm  := bInternalAlarm_b200_01_CircTankCircPumpTORAlarm ;
		DS_Alarm.b200_02_ThermalOilPumpTORAlarm  := bInternalAlarm_b200_02_ThermalOilPumpTORAlarm ;
		DS_Alarm.b200_03_ThermalOilLowLevelAlarm  := bInternalAlarm_b200_03_ThermalOilLowLevelAlarm ;
		DS_Alarm.b200_04_ThermalOilTempHighAlarm  := bInternalAlarm_b200_04_ThermalOilTempHighAlarm ;
		DS_Alarm.b200_05_ThermalOilTempNotReadyAlarm  := bInternalAlarm_b200_05_ThermalOilTempNotReadyAlarm ;
		DS_Alarm.b200_06_ThermalOilHeaterOnOffAlarm  := bInternalAlarm_b200_06_ThermalOilHeaterOnOffAlarm ;
		DS_Alarm.b200_07_TopDistillatorTempHighAlarm  := bInternalAlarm_b200_07_TopDistillatorTempHighAlarm ;
		DS_Alarm.b200_08_TopDistillatorTempNotReadyAlarm  := bInternalAlarm_b200_08_TopDistillatorTempNotReadyAlarm ;
		DS_Alarm.b200_09_TopDistillatorHeaterOnOffAlarm  := bInternalAlarm_b200_09_TopDistillatorHeaterOnOffAlarm ;
		DS_Alarm.b200_10_RecycleStartStopPBAlarm  := bInternalAlarm_b200_10_RecycleStartStopPBAlarm ;
		DS_Alarm.b200_11_EstopPBAlarm  := bInternalAlarm_b200_11_EstopPBAlarm ;

		DS_Alarm.b201_00_PhaseSeqenceRelayAlarm  := bInternalAlarm_b201_00_PhaseSeqenceRelayAlarm ;
		DS_Alarm.b201_01_ThermalOilUpThermostatAlarm  := bInternalAlarm_b201_01_ThermalOilUpThermostatAlarm ;
		DS_Alarm.b201_02_SludgeTankHighLevelAlarm  := bInternalAlarm_b201_02_SludgeTankHighLevelAlarm ;
		DS_Alarm.b201_03_FreshHCTankLowLevelAlarm  := bInternalAlarm_b201_03_FreshHCTankLowLevelAlarm ;
		DS_Alarm.b201_04_VacuumNotAchieveAlarm  := bInternalAlarm_b201_04_VacuumNotAchieveAlarm ;
		DS_Alarm.b201_05_IncomingCDALowPressureAlarm  := bInternalAlarm_b201_05_IncomingCDALowPressureAlarm ;
		DS_Alarm.b201_06_CoolingWaterLowFlowAlarm  := bInternalAlarm_b201_06_CoolingWaterLowFlowAlarm ;
		DS_Alarm.b201_07_CircularTankLowLevelAlarm  := bInternalAlarm_b201_07_CircularTankLowLevelAlarm ;
		DS_Alarm.b201_08_BottomDistillatorTempHighAlarm  := bInternalAlarm_b201_08_BottomDistillatorTempHighAlarm ;
		DS_Alarm.b201_09_BottomDistillatorTempNotReadyAlarm  := bInternalAlarm_b201_09_BottomDistillatorTempNotReadyAlarm ;
		DS_Alarm.b201_10_BottomDistillatorHeaterOnOffAlarm  := bInternalAlarm_b201_10_BottomDistillatorHeaterOnOffAlarm ;
		DS_Alarm.b201_11_ThermalOilDownThermostatAlarm  := bInternalAlarm_b201_11_ThermalOilDownThermostatAlarm ;
		DS_Alarm.b201_12_ThermalOilMidThermostatAlarm  := bInternalAlarm_b201_12_ThermalOilMidThermostatAlarm ;

		DS_Alarm.b202_00_VaporGenerationTempHighAlarm  := bInternalAlarm_b202_00_VaporGenerationTempHighAlarm ;
		DS_Alarm.b202_01_VaporGenerationTempNotReadyAlarm  := bInternalAlarm_b202_01_VaporGenerationTempNotReadyAlarm ;
		DS_Alarm.b202_02_VaporGenerationHeaterOnOffAlarm  := bInternalAlarm_b202_02_VaporGenerationHeaterOnOffAlarm ;
		DS_Alarm.b202_03_WasteCollectionTankLowLevelAlarm  := bInternalAlarm_b202_03_WasteCollectionTankLowLevelAlarm ;
		DS_Alarm.b202_04_VaporGenerationTankLowLevelAlarm  := bInternalAlarm_b202_04_VaporGenerationTankLowLevelAlarm ;
		DS_Alarm.b202_05_HCPurgingAV3_1Alarm  := bInternalAlarm_b202_05_HCPurgingAV3_1Alarm ;
		DS_Alarm.b202_06_MainMachineWasteTankLowLevelAlarm  := bInternalAlarm_b202_06_MainMachineWasteTankLowLevelAlarm ;
		DS_Alarm.b202_07_MainMachineWasteTankHighLevelAlarm  := bInternalAlarm_b202_07_MainMachineWasteTankHighLevelAlarm ;
		DS_Alarm.b202_08_ReservedAlarm  := bInternalAlarm_b202_08_ReservedAlarm ;
		DS_Alarm.b202_09_ReservedAlarm  := bInternalAlarm_b202_09_ReservedAlarm ;
		DS_Alarm.b202_10_ReservedAlarm  := bInternalAlarm_b202_10_ReservedAlarm ;
		DS_Alarm.b202_11_ReservedAlarm  := bInternalAlarm_b202_11_ReservedAlarm ;
		
		DS_Alarm.b203_00_ChillerSelectorOnOffAlarm  := bInternalAlarm_b203_00_ChillerSelectorOnOffAlarm ;
		DS_Alarm.b203_01_ColdWaterTankLowLevelAlarm  := bInternalAlarm_b203_01_ColdWaterTankLowLevelAlarm ;
		DS_Alarm.b203_02_SludgeTankMissingAlarm  := bInternalAlarm_b203_02_SludgeTankMissingAlarm ;
		DS_Alarm.b203_03_ColdWaterTankTempHighAlarm  := bInternalAlarm_b203_03_ColdWaterTankTempHighAlarm ;
		DS_Alarm.b203_04_ColdWaterTankTempNotReadyAlarm  := bInternalAlarm_b203_04_ColdWaterTankTempNotReadyAlarm ;
		DS_Alarm.b203_05_ColdWaterTankHeaterOnOffAlarm  := bInternalAlarm_b203_05_ColdWaterTankHeaterOnOffAlarm ;
		DS_Alarm.b203_06_ChillerPumpTORAlarm  := bInternalAlarm_b203_06_ChillerPumpTORAlarm ;
		DS_Alarm.b203_07_ChillerFlowSwitchAlarm  := bInternalAlarm_b203_07_ChillerFlowSwitchAlarm ;
		DS_Alarm.b203_08_ChillerInterlockRelayAlarm  := bInternalAlarm_b203_08_ChillerInterlockRelayAlarm ;
		DS_Alarm.b203_09_ReservedAlarm  := bInternalAlarm_b203_09_ReservedAlarm ;
		DS_Alarm.b203_10_ThermalOilChangeWarning  := bInternalAlarm_b203_10_ThermalOilChangeWarning ;
		DS_Alarm.b203_11_ThermalOilChangeAlarm  := bInternalAlarm_b203_11_ThermalOilChangeAlarm ;
		
		
		(*Mapping - Input*)	
		bInternalInput_b000_00_FreshHCTankCircPumpTOR  := DS_Input.b000_00_FreshHCTankCircPumpTOR ;
		bInternalInput_b000_01_CircTankCircPumpTOR  := DS_Input.b000_01_CircTankCircPumpTOR ;
		bInternalInput_b000_02_ThermalOilPumpTOR := DS_Input.b000_02_ThermalOilPumpTOR;
		bInternalInput_b000_03_ThermalOilLevelSensor := DS_Input.b000_03_ThermalOilLevelSensor;
(*		bInternalInput_b000_04_ThermalOilTempCtrlHighTempAlarmSignal := DS_Input.b000_04_ThermalOilTempCtrlHighTempAlarmSignal;
		bInternalInput_b000_05_ThermalOilTempCtrlReadySignal := DS_Input.b000_05_ThermalOilTempCtrlReadySignal;
		bInternalInput_b000_06_ThermalOilTempCtrlOnOffSignal  := DS_Input.b000_06_ThermalOilTempCtrlOnOffSignal ;
		bInternalInput_b000_07_TopDistillatorTempCtrlHighTempAlarmSignal := DS_Input.b000_07_TopDistillatorTempCtrlHighTempAlarmSignal;
		bInternalInput_b000_08_TopDistillatorTempCtrlReadySignal := DS_Input.b000_08_TopDistillatorTempCtrlReadySignal;
		bInternalInput_b000_09_TopDistillatorTempCtrlOnOffSignal  := DS_Input.b000_09_TopDistillatorTempCtrlOnOffSignal ;
*)		bInternalInput_b000_10_RecycleStartStopPB := DS_Input.b000_10_RecycleStartStopPB;
		bInternalInput_b000_11_EStopPB := DS_Input.b000_11_EStopPB;


		bInternalInput_b001_00_PhaseSequenceRelayAlarm := DS_Input.b001_00_PhaseSequenceRelayAlarm;
		bInternalInput_b001_01_ThermalOilUpThermostat  := DS_Input.b001_01_ThermalOilUpThermostat ;
		bInternalInput_b001_02_SludgeTankLevelSensor := DS_Input.b001_02_SludgeTankLevelSensor;
		bInternalInput_b001_03_FreshHCTankLevelSensor := DS_Input.b001_03_FreshHCTankLevelSensor;
(*		bInternalInput_b001_04_VacuumNotAchieveSignal := DS_Input.b001_04_VacuumNotAchieveSignal;
*)		bInternalInput_b001_05_IncomingCDAPressureSwitch := DS_Input.b001_05_IncomingCDAPressureSwitch;
		bInternalInput_b001_06_CoolingWaterFlowSwitch := DS_Input.b001_06_CoolingWaterFlowSwitch;
		bInternalInput_b001_07_CircularTankLevelSensor := DS_Input.b001_07_CircularTankLevelSensor;
(*		bInternalInput_b001_08_BottomDistillatorTempCtrlHighTempAlarmSignal := DS_Input.b001_08_BottomDistillatorTempCtrlHighTempAlarmSignal;
		bInternalInput_b001_09_BottomDistillatorTempCtrlReadySignal := DS_Input.b001_09_BottomDistillatorTempCtrlReadySignal;
		bInternalInput_b001_10_BottomDistillatorTempCtrlOnOffSignal  := DS_Input.b001_10_BottomDistillatorTempCtrlOnOffSignal ;
*)		bInternalInput_b001_11_ThermalOilDownThermostat := DS_Input.b001_11_ThermalOilDownThermostat;
		bInternalInput_b001_12_ThermalOilMidThermostat := DS_Input.b001_12_ThermalOilMidThermostat;

(*		bInternalInput_b002_00_VaporGenerationTempCtrlHighTempAlarmSignal := DS_Input.b002_00_VaporGenerationTempCtrlHighTempAlarmSignal;
		bInternalInput_b002_01_VaporGenerationTempCtrlReadySignal := DS_Input.b002_01_VaporGenerationTempCtrlReadySignal;
		bInternalInput_b002_02_VaporGenerationTempCtrlOnOffSignal := DS_Input.b002_02_VaporGenerationTempCtrlOnOffSignal;
*)		bInternalInput_b002_03_WasteCollectionTankLevelSensor := DS_Input.b002_03_WasteCollectionTankLevelSensor;
		bInternalInput_b002_04_VaporGenerationTankLowLevelSensor := DS_Input.b002_04_VaporGenerationTankLowLevelSensor;
		bInternalInput_b002_05_HCPurgingAV := DS_Input.b002_05_HCPurgingAV;
		bInternalInput_b002_06_MainMachineWasteCollectTankLowLevelSignal := DS_Input.b002_06_MainMachineWasteCollectTankLowLevelSignal;
		bInternalInput_b002_07_MainMachineWasteCollectTankHighLevelSignal := DS_Input.b002_07_MainMachineWasteCollectTankHighLevelSignal;
		bInternalInput_b002_08_FromMainMachineSignal3 := DS_Input.b002_08_FromMainMachineSignal3;
		bInternalInput_b002_09_FromMainMachineSignal4 := DS_Input.b002_09_FromMainMachineSignal4;
		bInternalInput_b002_10_FromMainMachineSignal5 := DS_Input.b002_10_FromMainMachineSignal5;
		bInternalInput_b002_11_ReservedAlarmSignal := DS_Input.b002_11_ReservedAlarmSignal;


		bInternalInput_b003_00_ChillerSelectorOnOff := DS_Input.b003_00_ChillerSelectorOnOff;
		bInternalInput_b003_01_ColdWaterTankLowLevelSensor := DS_Input.b003_01_ColdWaterTankLowLevelSensor;
		bInternalInput_b003_02_SludgeTankPresentSensor := DS_Input.b003_02_SludgeTankPresentSensor;
(*		bInternalInput_b003_03_ColdWaterTankTempCtrlHighTempAlarmSignal := DS_Input.b003_03_ColdWaterTankTempCtrlHighTempAlarmSignal;
		bInternalInput_b003_04_ColdWaterTankTempCtrlReadySignal := DS_Input.b003_04_ColdWaterTankTempCtrlReadySignal;
		bInternalInput_b003_05_ColdWaterTankTempCtrlOnOffSignal := DS_Input.b003_05_ColdWaterTankTempCtrlOnOffSignal;
*)		bInternalInput_b003_06_ChillerPumpTOR := DS_Input.b003_06_ChillerPumpTOR;
		bInternalInput_b003_07_ChillerFlowSwitch := DS_Input.b003_07_ChillerFlowSwitch;
		bInternalInput_b003_08_ChillerInterlockRelay := DS_Input.b003_08_ChillerInterlockRelay;
		bInternalInput_b003_09_ReservedAlarmSignal := DS_Input.b003_09_ReservedAlarmSignal;
		bInternalInput_b003_10_ReservedAlarmSignal := DS_Input.b003_10_ReservedAlarmSignal;
		bInternalInput_b003_11_ReservedAlarmSignal := DS_Input.b003_11_ReservedAlarmSignal;
		
		(*Mapping - Output*)
		DS_Output.b100_00_FreshHCTankCircPumpOnOff  := bInternalOutput_b100_00_FreshHCTankCircPumpOnOff ;
		DS_Output.b100_01_CircTankCircPumpOnOff := bInternalOutput_b100_01_CircTankCircPumpOnOff;
		DS_Output.b100_02_ThermalOilPumpOnOff := bInternalOutput_b100_02_ThermalOilPumpOnOff;
		DS_Output.b100_03_ThermalOilHeaterOnOff := bInternalOutput_b100_03_ThermalOilHeaterOnOff;
		DS_Output.b100_04_Buzzer := bInternalOutput_b100_04_Buzzer;
		DS_Output.b100_05_RecycleStartStopIndicator := bInternalOutput_b100_05_RecycleStartStopIndicator;
		DS_Output.b100_06_Reserved := bInternalOutput_b100_06_Reserved;
		DS_Output.b100_07_UFOVacuumRelease32WayAV := bInternalOutput_b100_07_UFOVacuumRelease32WayAV;
		
		
		DS_Output.b101_00_CondenserTankVacuumReleaseAV := bInternalOutput_b101_00_CondenserTankVacuumReleaseAV;
		DS_Output.b101_01_WasteSludgeCollectionDrumAV  := bInternalOutput_b101_01_WasteSludgeCollectionDrumAV ;
		DS_Output.b101_02_DistillationTankDrainAV := bInternalOutput_b101_02_DistillationTankDrainAV;
		DS_Output.b101_03_EconomizerAV := bInternalOutput_b101_03_EconomizerAV;
		DS_Output.b101_04_Reserved := bInternalOutput_b101_04_Reserved;
		DS_Output.b101_05_Reserved := bInternalOutput_b101_05_Reserved;
		DS_Output.b101_06_VaporGenerationAV := bInternalOutput_b101_06_VaporGenerationAV;
		DS_Output.b101_07_VacuumSharingAV := bInternalOutput_b101_07_VacuumSharingAV;

		
		DS_Output.b102_00_RecycleReadySignal := bInternalOutput_b102_00_RecycleReadySignal;
		DS_Output.b102_01_VaporNotAvailableForRequestSignal := bInternalOutput_b102_01_VaporNotAvailableForRequestSignal;
		DS_Output.b102_02_ToMainMachineSignal3 := bInternalOutput_b102_02_ToMainMachineSignal3;
		DS_Output.b102_03_ToMainMachineSignal4 := bInternalOutput_b102_03_ToMainMachineSignal4;
		DS_Output.b102_04_ToMainMachineSignal5 := bInternalOutput_b102_04_ToMainMachineSignal5;
		DS_Output.b102_05_Reserved := bInternalOutput_b102_05_Reserved;
		DS_Output.b102_06_Reserved := bInternalOutput_b102_06_Reserved;
		DS_Output.b102_07_Reserved := bInternalOutput_b102_07_Reserved;
		
		
		DS_Output.b103_00_ChillerPumpOnOff := bInternalOutput_b103_00_ChillerPumpOnOff;
		DS_Output.b103_01_Reserved := bInternalOutput_b103_01_Reserved;
		DS_Output.b103_02_Reserved := bInternalOutput_b103_02_Reserved;
		DS_Output.b103_03_Reserved := bInternalOutput_b103_03_Reserved;
		DS_Output.b103_04_ChillerSelectorOnOffIndicator := bInternalOutput_b103_04_ChillerSelectorOnOffIndicator;
		DS_Output.b103_05_ChillerReadySignal := bInternalOutput_b103_05_ChillerReadySignal;
		DS_Output.b103_06_ChillerCompressorOnOff := bInternalOutput_b103_06_ChillerCompressorOnOff;
		DS_Output.b103_07_Reserved := bInternalOutput_b103_07_Reserved;
END_ACTION

END_FUNCTION_BLOCK

(* stored: Version 1.1.0.1, ProductVersion 3.1.4024.12
   POU fb_V3JRSModuleWithChiller: Id {8de57156-a313-4887-b3c6-7e2376d45017}, SpecialFunc None
   Action AlarmCtrl_LD: Id {658a0a97-7752-40bd-b394-33bd238a50fb}
   Action AutoBoilingCtrl_LD: Id {44a33cae-4785-4eeb-8770-d1e7941e1337}
   Action AutoBoilingCtrl_ST: Id {08eb34b8-944f-4bad-b752-df8f47d8906d}
   Action AutoCtrl_LD: Id {f289761c-db85-4887-ad06-3e07f0987822}
   Action AutoHCTopUp_LD: Id {050e1469-a41a-467a-b9a9-94191b0fdbe9}
   Action BuzzerCtrl_ST: Id {6fce0cdf-0011-4b68-a60f-9b78ae694650}
   Action ChillerCtrl_LD: Id {d1f24c9f-353a-475e-b288-6bddfb71a0fa}
   Action FixOutput_LD: Id {369e373e-42dc-4983-aabf-5c407a2d4925}
   Action HighLowLimitCtrl_ST: Id {44b080d9-602e-420f-bced-fa83e09bbefd}
   Action JRSMachineServiceCtrl_LD: Id {20f18914-3de3-485a-91bb-1115ccd94e04}
   Action ManualBoilingCtrl_LD: Id {3d5478e3-dd7d-4c74-b5a5-6e3c5f7b70e8}
   Action ManualBoilingCtrl_ST: Id {1bf449df-b5fa-4eb5-89bc-dafe54a29424}
   Action ManualCtrl_ST: Id {2f958cdd-7dd2-4a70-b913-4fe924693d7f}
   Action MessageDisplayCtrl_ST: Id {98b38ef8-108a-475f-b8f8-17bb5854cf9e}
   Action Other_LD: Id {5abe569f-491c-4882-9a55-d965061e157b}
   Action Other_ST: Id {f05cb890-2a54-4b74-9726-bab0d47c119b}
   Action OutputCtrl_LD: Id {1ba9302a-3759-4e93-af88-61775efad123}
   Action SystemRestore_LD: Id {3c08baa0-0c19-4de0-8844-23e5963254bd}
   Action ThermalOilChangeHRMeter_ST: Id {c3e4ba57-15c4-43e6-8e0f-ffa6e6f0a596}
   Action Z_BuiltInTempCtrl_LD: Id {54cc019b-1cc8-4c95-9ec1-f37d5f753b27}
   Action Z_BuiltInTempCtrl_ST: Id {f3fb7ccc-d1b0-4eaf-b5a0-39a364fa0688}
   Action Z_BuiltInVacuumCtrl_LD: Id {a7c5e23a-06b8-4fe2-ae3b-1dd6adb705ab}
   Action Z_BuiltInVacuumCtrl_ST: Id {7d709ef2-25fe-4301-a39a-2a41858f8d25}
   Action Z_Mapping: Id {90838cb2-d650-400e-8253-aad89bde7f95} *)
